// TwinCAT 3 PLC project AddDataToDB
// ProgramVersion: 3.1.4024.0
// libraries:
//   Tc2_IoFunctions, * (Beckhoff Automation GmbH)
//   Tc2_Standard, * (Beckhoff Automation GmbH)
//   Tc2_System, * (Beckhoff Automation GmbH)
//   Tc2_Utilities, * (Beckhoff Automation GmbH)
//   Tc3_Database, * (Beckhoff Automation GmbH)
//   Tc3_Module, * (Beckhoff Automation GmbH)
// project tree:
//   GVLs/ GVL.TcGVL
//   / PlcTask.TcTTO
//   POUs/ DBSync.TcPOU, MAIN.TcPOU, PeriodicMesure.TcPOU, POU.TcPOU, pTimer.TcPOU
// real-time tasks:
//   TASK PlcTask: cycle T#10ms, priority 20, ADS port 350
// I/O:
//   DEVICE Device 2 (EtherCAT), AmsNetId 172.18.233.216.3.1
//     Term 1 (EK1100) [EK1100 EtherCAT Coupler (2A E-Bus)]
//       Term 2 (EL2014) [EL2014 4Ch. Dig. Output 24V, 0,5A, Diagnostic]
//       Term 3 (EL3124) [EL3124 4Ch. Ana. Input 4-20mA Diff.]
//       Term 4 (EL9011) [EL9011 End Terminal]
// variable links:
//   AddDataToDB/AddDataToDB Instance <-> Device 2 (EtherCAT)/Term 1 (EK1100)/Term 2 (EL2014)
//     PlcTask Outputs/GVL.bVR20On <-> DIG Outputs/Channel 2/Output
//     PlcTask Outputs/GVL.bVR25On <-> DIG Outputs/Channel 1/Output
//   AddDataToDB/AddDataToDB Instance <-> Device 2 (EtherCAT)/Term 1 (EK1100)/Term 3 (EL3124)
//     PlcTask Inputs/GVL.iVR20Value <-> AI Standard Channel 2/Value
//     PlcTask Inputs/GVL.iVR25Value <-> AI Standard Channel 1/Value

CONFIGURATION AddDataToDB
    RESOURCE PLC ON TwinCAT3
        TASK PlcTask(INTERVAL := T#10ms, PRIORITY := 20);
        PROGRAM MAIN WITH PlcTask : MAIN;
    END_RESOURCE
END_CONFIGURATION

// ---- GVLs/GVL.TcGVL
{attribute 'qualified_only'}
VAR_GLOBAL
	bVR25On AT %Q* : BOOL := TRUE; // Switch on/off capteur VR25
	bVR20On AT %Q* : BOOL := TRUE; // Switch on/off capteur VR20
	
	iVR25Value AT %I* : INT; // Valeur Brute VR25 depuis EL3124
	iVR20Value AT %I* : INT; // Valeur Brute VR20 depuis EL3124
	
	iIDClient : INT := 1; // ID Client dans BDD
	
	iIDPlant : INT := 1; // ID Plant dans BDD
	
	iIDMachine : INT := 1; // ID Machine dans BDD
	
	iIDImageVR25 : INT := 1; // ID Image VR25 dans BDD
	iIDImageVR20 : INT := 2; // ID Image VR20 dans BDD
	
	iIDDAQVR25 : INT := 1; // ID DAQ VR25 dans BDD
	iIDDAQVR20 : INT := 2; // ID DAQ VR20 dans BDD
	
	sTypeVR25 : STRING := 'Acceleration'; // Type de mesure par VR25 dans JSON
	sTypeVR20 : STRING := 'Acceleration'; // Type de mesure par VR20 dans JSON
	
	sUomVR25 : STRING := 'mm/s'; // Unité de mesure par VR25 dans JSON
	sUomVR20 : STRING := 'mm/s'; // Unité de mesure par VR20 dans JSON
	
END_VAR

// ---- POUs/MAIN.TcPOU
PROGRAM MAIN
VAR
	bStartExport : BOOL;
	bStartImport : BOOL;
	bStartAquisition : BOOL;
END_VAR

IF bStartExport THEN
	bStartExport := FALSE;
	DBSync(bExportTrigger := TRUE);
ELSIF bStartImport THEN
	bStartImport := FALSE;
	DBSync(bImportTrigger := TRUE);
ELSIF bStartAquisition THEN
	pTimer();
END_IF

END_PROGRAM

// ---- POUs/DBSync.TcPOU
PROGRAM DBSync
VAR_INPUT
	bExportTrigger : BOOL ;
	bImportTrigger : BOOL ;
END_VAR
VAR
	Process : NT_StartProcess;

    bError : BOOL;
    iErrorId : UDINT;
	bIsBusy : BOOL;
END_VAR

IF bExportTrigger THEN
	Process(
    	NETID := '', 
    	PATHSTR := 'C:\Windows\System32\cmd.exe',  
		COMNDLINE := '/C start cmd /c C:\Users\Administrator\Documents\Scripts\Export.cmd',
		TMOUT := T#1M,
    	ERR => bError,            
    	ERRID => iErrorId,
		BUSY => bIsBusy       
	);
	
	
	Process(START:=TRUE);
    Process(START:=FALSE);
    bExportTrigger := FALSE;
	
ELSIF bImportTrigger THEN
	Process(
    	NETID := '', 
    	PATHSTR := 'C:\Windows\System32\cmd.exe',
    	COMNDLINE := '/C start cmd /c C:\Users\Administrator\Documents\Scripts\Import.cmd',      
    	ERR => bError,            
    	ERRID => iErrorId           
	);
    bImportTrigger := FALSE;
    Process(START:=TRUE);
    Process(START:=FALSE);
	
END_IF

END_PROGRAM

// ---- POUs/pTimer.TcPOU
PROGRAM pTimer
VAR_INPUT
	timer : TON;
END_VAR

timer(IN := TRUE, PT := T#5S);
IF timer.Q THEN
	PeriodicMesure();
	timer(IN := NOT PeriodicMesure.isfinished());
END_IF

END_PROGRAM

// ---- POUs/PeriodicMesure.TcPOU
PROGRAM PeriodicMesure
VAR
	fbSQLDatabase : FB_SQLDatabaseEvt(sNetID := '', tTimeout := T#5S);

	fbSQLCommand : FB_SQLCommandEvt(sNetID := '', tTimeOut := T#5S);

	step : (OPEN_CONNECTION, CREATE_MESURE, INSERT_MESURE, CLOSE_CONNECTION, FINISH) := OPEN_CONNECTION;
	CMD25 : STRING(255);
	CMD20 : STRING(255);
	CMD : STRING(1000);
	
	rVR25True : REAL;
	rVR20True : REAL;
	
	jsonString : STRING(5000);
	
	
END_VAR

CASE step OF
	
	OPEN_CONNECTION:

		IF fbSQLDatabase.Connect(1) THEN
			step := CREATE_MESURE;
		END_IF
		
	CREATE_MESURE:
		IF fbSQLDatabase.CreateCmd(ADR(fbSQLCommand)) THEN
			step := INSERT_MESURE;
		END_IF
		
	INSERT_MESURE:
		
		// Convert raw value to mm/s
	
		rVR25True := GVL.iVR25Value * 0.000488296151 * 1.5625;
		rVR20True := GVL.iVR20Value * 0.000488296151 * 1.25;
		
		// Creating jsonString VR25
		
		jsonString := CONCAT('$'{"type":"', GVL.sTypeVR25);
		jsonString := CONCAT(jsonString, '","uom":"');
		jsonString := CONCAT(jsonString, GVL.sUomVR25);
		jsonString := CONCAT(jsonString, '","value":');
		jsonString := CONCAT(jsonString, REAL_TO_STRING(rVR25True));
		jsonString := CONCAT(jsonString, '}$'');
		
		// Creating SQL Query VR25
	
		CMD25 := CONCAT('INSERT INTO Tag (timestampStart, json_data, id_client, id_machine, id_daq, id_plant, id_image) VALUES (',ULINT_TO_STRING(F_GetSystemTime()));
		CMD25 := CONCAT(CMD25, ',');
		CMD25 := CONCAT(CMD25, jsonString);
		CMD25 := CONCAT(CMD25, ',');
		CMD25 := CONCAT(CMD25, INT_TO_STRING(GVL.iIDClient));
		CMD25 := CONCAT(CMD25, ',');
		CMD25 := CONCAT(CMD25, INT_TO_STRING(GVL.iIDMachine));
		CMD25 := CONCAT(CMD25, ',');
		CMD25 := CONCAT(CMD25, INT_TO_STRING(GVL.iIDDAQVR25));
		CMD25 := CONCAT(CMD25, ',');
		CMD25 := CONCAT(CMD25, INT_TO_STRING(GVL.iIDPlant));
		CMD25 := CONCAT(CMD25, ',');
		CMD25 := CONCAT(CMD25, INT_TO_STRING(GVL.iIDImageVR25));
		CMD25 := CONCAT(CMD25, ');');
		
		// Creating jsonString VR20
		
		jsonString := CONCAT('$'{"type":"', GVL.sTypeVR20);
		jsonString := CONCAT(jsonString, '","uom":"');
		jsonString := CONCAT(jsonString, GVL.sUomVR20);
		jsonString := CONCAT(jsonString, '","value":');
		jsonString := CONCAT(jsonString, REAL_TO_STRING(rVR20True));
		jsonString := CONCAT(jsonString, '}$'');
		
		// Creating SQL Query VR20
		
		CMD20 := CONCAT('INSERT INTO Tag (timestampStart, json_data, id_client, id_machine, id_daq, id_plant, id_image) VALUES (',ULINT_TO_STRING(F_GetSystemTime()));
		CMD20 := CONCAT(CMD20, ',');
		CMD20 := CONCAT(CMD20, jsonString);
		CMD20 := CONCAT(CMD20, ',');
		CMD20 := CONCAT(CMD20, INT_TO_STRING(GVL.iIDClient));
		CMD20 := CONCAT(CMD20, ',');
		CMD20 := CONCAT(CMD20, INT_TO_STRING(GVL.iIDMachine));
		CMD20 := CONCAT(CMD20, ',');
		CMD20 := CONCAT(CMD20, INT_TO_STRING(GVL.iIDDAQVR20));
		CMD20 := CONCAT(CMD20, ',');
		CMD20 := CONCAT(CMD20, INT_TO_STRING(GVL.iIDPlant));
		CMD20 := CONCAT(CMD20, ',');
		CMD20 := CONCAT(CMD20, INT_TO_STRING(GVL.iIDImageVR20));
		CMD20 := CONCAT(CMD20, ');');
		
		CONCAT2(ADR(CMD25), ADR(CMD20), ADR(CMD), SIZEOF(CMD));
		
		IF fbSQLCommand.Execute(ADR(CMD), SIZEOF(CMD)) THEN
			step := CLOSE_CONNECTION;
		END_IF
	
	CLOSE_CONNECTION:
		IF fbSQLDatabase.Disconnect() THEN
			step := FINISH;
		END_IF
		
	FINISH:
		step := OPEN_CONNECTION; 

		
END_CASE

METHOD isfinished : BOOL
IF step = FINISH THEN
	isfinished := TRUE;
ELSE
	isfinished := FALSE;
END_IF
END_METHOD

END_PROGRAM

// ---- POUs/POU.TcPOU
FUNCTION StringAssembly : STRING

VAR_IN_OUT
	liste : ARRAY [*] OF WORD; 
END_VAR

VAR
	counter : INT;
END_VAR

END_FUNCTION
